// SIMATIC S7-200 project (STEP 7-Micro/WIN), CPU 221 REL 01.10

ORGANIZATION_BLOCK MAIN:OB1
TITLE=PROGRAM COMMENTS
BEGIN
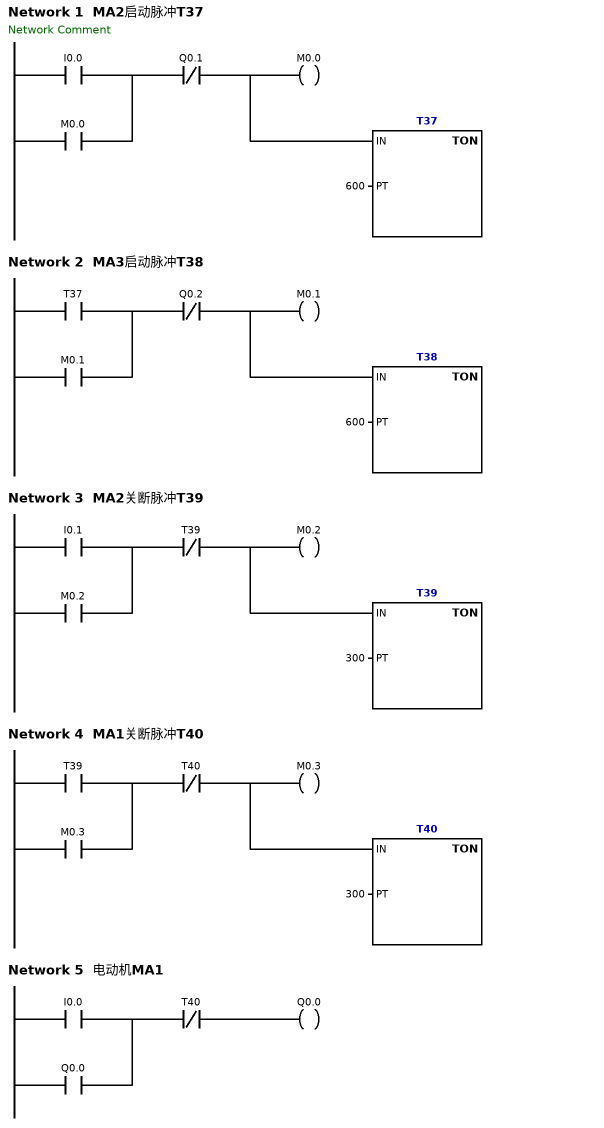
Network 1 // MA2启动脉冲T37
// Network Comment
// (network saved uncompiled; LAD cells follow)
// row 0: c0 -| |- I0.0 v  c1 -|/|- Q0.1 v  c2 -( ) M0.0
// row 1: c0 -| |- M0.0 ^  c1 ^  c2 --  c3 [TON T37 IN:=power@row1, PT:=600]
// row 2: c3 [box]
Network 2 // MA3启动脉冲T38
// (network saved uncompiled; LAD cells follow)
// row 0: c0 -| |- T37 v  c1 -|/|- Q0.2 v  c2 -( ) M0.1
// row 1: c0 -| |- M0.1 ^  c1 ^  c2 --  c3 [TON T38 IN:=power@row1, PT:=600]
// row 2: c3 [box]
Network 3 // MA2关断脉冲T39
// (network saved uncompiled; LAD cells follow)
// row 0: c0 -| |- I0.1 v  c1 -|/|- T39 v  c2 -( ) M0.2
// row 1: c0 -| |- M0.2 ^  c1 ^  c2 --  c3 [TON T39 IN:=power@row1, PT:=300]
// row 2: c3 [box]
Network 4 // MA1关断脉冲T40
// (network saved uncompiled; LAD cells follow)
// row 0: c0 -| |- T39 v  c1 -|/|- T40 v  c2 -( ) M0.3
// row 1: c0 -| |- M0.3 ^  c1 ^  c2 --  c3 [TON T40 IN:=power@row1, PT:=300]
// row 2: c3 [box]
Network 5 // 电动机MA1
// (network saved uncompiled; LAD cells follow)
// row 0: c0 -| |- I0.0 v  c1 -|/|- T40  c2 -( ) Q0.0
// row 1: c0 -| |- Q0.0 ^
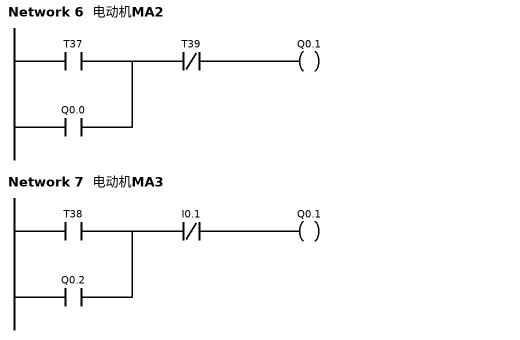
Network 6 // 电动机MA2
// (network saved uncompiled; LAD cells follow)
// row 0: c0 -| |- T37 v  c1 -|/|- T39  c2 -( ) Q0.1
// row 1: c0 -| |- Q0.0 ^
Network 7 // 电动机MA3
// (network saved uncompiled; LAD cells follow)
// row 0: c0 -| |- T38 v  c1 -|/|- I0.1  c2 -( ) Q0.1
// row 1: c0 -| |- Q0.2 ^
END_ORGANIZATION_BLOCK
